FUNCTION_BLOCK Monitor
  (* Standard: 61499-2 *)
  (* Version 0.2, 2003-12-04, JHC, Rockwell Automation, Renamed for better indexing. *)
  (* Version 0.1, 2002-11-05, JHC, Rockwell Automation, Corrected missing ST element in Algorithm REQ. *)
  (* Version 0.0, 2000-05-30, JHC, Rockwell Automation *)
  (* Compiler header: package fb.rt.benchmarks.watermonitor; *)
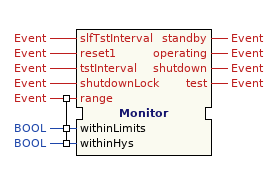
  EVENT_INPUT
    slfTstInterval;
    reset1;
    tstInterval;
    shutdownLock;
    range WITH withinLimits, withinHys;
  END_EVENT
  EVENT_OUTPUT
    standby;
    operating;
    shutdown;
    test;
  END_EVENT
  VAR_INPUT
    withinLimits : BOOL := true;
    withinHys : BOOL := true;
  END_VAR
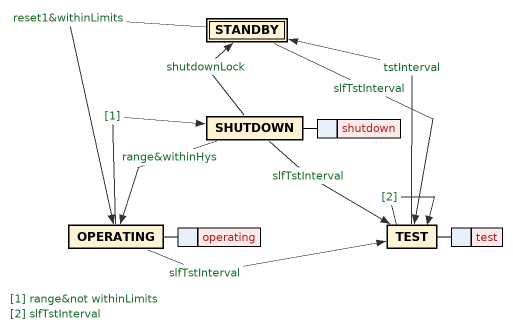
  EC_STATES
    STANDBY; (* Initial State *)
    SHUTDOWN : -> shutdown;
    OPERATING : -> operating;
    TEST : -> test;
  END_STATES
  EC_TRANSITIONS
    STANDBY TO TEST := slfTstInterval;
    STANDBY TO OPERATING := reset1&withinLimits;
    TEST TO TEST := slfTstInterval;
    TEST TO STANDBY := tstInterval;
    OPERATING TO TEST := slfTstInterval;
    OPERATING TO SHUTDOWN := range&not withinLimits;
    SHUTDOWN TO TEST := slfTstInterval;
    SHUTDOWN TO OPERATING := range&withinHys;
    SHUTDOWN TO STANDBY := shutdownLock;
  END_TRANSITIONS
END_FUNCTION_BLOCK
